TYPE iol_slave_mlg2prime_system_status_1 :
STRUCT
	sync_error:					BIT;
	teach_fail:					BIT;
	hardware_error:				BIT;
	contamination_alarm:		BIT;
	teach_active:				BIT;
	over_temp:					BIT;
	data_invalid:				BIT;
	q_short_circuit:			BIT;
END_STRUCT
END_TYPE

(* stored: Version 1.1.0.1, ProductVersion 3.1.4024.3
   DUT iol_slave_mlg2prime_system_status_1: Id {faed7c66-216f-032f-2b6d-8114d13dc573} *)
